// TIA Portal V17 export
// export: Created 2025-06-25T13:13:10.2862432Z, ExportSetting WithDefaults, DisplayName Totally Integrated Automation Portal, DisplayVersion V17 Update 8, DisplayName TIA Portal Openness, DisplayVersion V17 Update 8, DisplayName TIA Portal Version Control Interface, DisplayVersion V17, DisplayName STEP 7 Professional, DisplayVersion V17 Update 8, DisplayName STEP 7 Safety, DisplayVersion V17 Update 6, DisplayName WinCC Advanced, DisplayVersion V17 Update 8
FUNCTION "ConsumedPower" : Void   // FC20, FBD
TITLE = Tally up consumers
{ S7_Optimized_Access := 'TRUE' }
VERSION : 0.1
// stored: AutoNumber true, IsIECCheckEnabled false, SetENOAutomatically false, UDAEnableTagReadback false
   VAR_TEMP
      fPower : Real;
   END_VAR
   VAR CONSTANT
      SSC_P_01_POWER : Real := 0.55;   // kW
      SSC_P_02_POWER : Real := 0.55;   // kW
      SSC_F_01_POWER : Real := 0.55;   // kW
      CPC_P_01_POWER : Real := 1.1;   // kW
      CabinetHeater_POWER : Real := 0.045;   // kW
      CabinetFan_POWER : Real := 0.1;   // kW
      HBL_EC_01_POWER : Real := 4.0;   // kW
      HBL_EC_02_POWER : Real := 8.0;   // kW
   END_VAR
BEGIN

REGION Network 1 (SCL)
   // Inverters. Do not convert to ELSIF
   IF "DB_InverterDrives".CPC_SC_01.Stat.Power.Eng.bError = FALSE THEN
       #fPower += "DB_InverterDrives".CPC_SC_01.Stat.Power.Eng.fValue;
   END_IF;
   IF "DB_InverterDrives".HBL_SC_01.Stat.Power.Eng.bError = FALSE THEN
       #fPower += "DB_InverterDrives".HBL_SC_01.Stat.Power.Eng.fValue;
   END_IF;
   IF "DB_InverterDrives".HBL_SC_02.Stat.Power.Eng.bError = FALSE THEN
       #fPower += "DB_InverterDrives".HBL_SC_02.Stat.Power.Eng.fValue;
   END_IF;
   IF "DB_InverterDrives".HBL_SC_10.Stat.Power.Eng.bError = FALSE THEN
       #fPower += "DB_InverterDrives".HBL_SC_10.Stat.Power.Eng.fValue;
   END_IF;

   // Auxiliary Motors. Do not convert to ELSIF
   IF "DB_DO".SSC_P_01 = TRUE THEN
       #fPower += #SSC_P_01_POWER;
   END_IF;
   IF "DB_DO".SSC_P_02 = TRUE THEN
       #fPower += #SSC_P_02_POWER;
   END_IF;
   IF "DB_DO".SSC_F_01 = TRUE THEN
       #fPower += #SSC_F_01_POWER;
   END_IF;
   IF "DB_DO".CPC_P_01 = TRUE THEN
       #fPower += #CPC_P_01_POWER;
   END_IF;

   // Cabinet heating & cooling. Do not convert to ELSIF
   IF "DB_DO".CabinetHeater = TRUE THEN
       #fPower += #CabinetHeater_POWER;
   END_IF;
   IF "DB_DO".CabinetFan = TRUE THEN
       #fPower += #CabinetHeater_POWER;
   END_IF;

   // Crankcase oil heaters. Do not convert to ELSIF
   IF "DB_DO".HBL_EC_01 = TRUE THEN
       #fPower += #HBL_EC_01_POWER;
   END_IF;
   IF "DB_DO".HBL_EC_02 = TRUE THEN
       #fPower += #HBL_EC_02_POWER;
   END_IF;

   // Store in calc object
   "fcCalcAssign"(fValue := #fPower, sTag := "DB_Calc".System.ElectricalPower);
END_REGION
END_FUNCTION
